Fanuc KAREL source: KD00010.KL

PROGRAM KD00010
%NOLOCKGROUP
%INCLUDE KDOCINC
VAR
  I: INTEGER
  J: INTEGER
  B: BOOLEAN
  R: REAL
  S: STRING[80]
BEGIN
  I = 1
END KD00010
